Universal Robots PolyScope program: space invade.urp

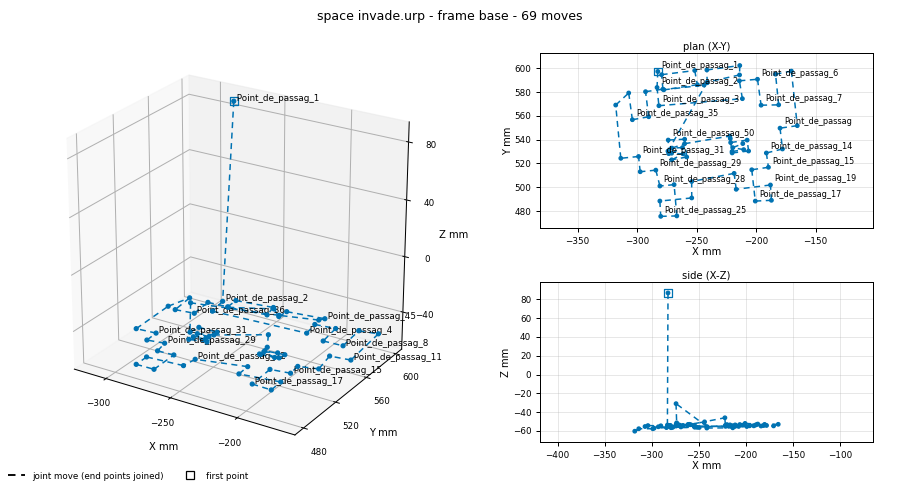
[picture p0: tool path of space invade.urp in frame base, 69 of 69 moves have a stored position in this frame; points joined in program order, loops and branches not executed]
ProgramRoot directory=/programs; kinematics=(a=[0, -0.425, -0.39225, 0, 0, 0], d=[0.08916, 0, 0, 0.10915, 0.09465, 0.0823], alpha=[1.5708, 0, 0, 1.5708, -1.5708, 0], deltaTheta=[0, 0, 0, 0, 0, 0], status=notInitialized); name=space invade; programVersion=(project__name=PolyScope, major__version=1, minor__version=6, svn__revision=9671, build__date=Dec 17 2012, 15:17:18); robotEnvironmentFileName=default
  MainProgram cartesianAcceleration=1.2; cartesianSpeed=0.25; jointAcceleration=1.3962634015954636; jointSpeed=1.0471975511965976; moveAsFastAsPossible=true; sharedProcessMoveBlendRadius=0.025; featureReference=(installationNameReference=Base); motionType=JOINT_SPACE
    Move cartesianAcceleration=1.2; cartesianSpeed=0.25; jointAcceleration=3.141592653589793; jointSpeed=3.2; moveAsFastAsPossible=true; sharedProcessMoveBlendRadius=0.025; featureReference=(installationNameReference=Base); motionType=JOINT_SPACE
      Waypoint blendRadius=0.05; cartesianAcceleration=1.2; cartesianSpeed=0.25; jointAcceleration=1.3962634015954636; jointSpeed=1.0471975511965976; nextMotionTime=2.0; stoppoint=true; useSharedBlendParameter=true; useSharedParameters=true; position=TCP in base x=-282.652 y=597.285 z=86.76 mm, rx=0.0179 ry=-1.8099 rz=-2.292 rad; joints [-73.183, -51.912, 94.402, -56.585, 97.955, 5.493] deg; positionType=FIXED_POSITION; waypointPoseInFeatureCoordinates=(pos=(x=-0.28265202221526026, y=0.5972847385628794, z=0.08675977077379672), rot=(x=0.017936265921650735, y=-1.8098588398059938, z=-2.292012778294841)); name=Point_de_passag_1
      Waypoint blendRadius=0.05; cartesianAcceleration=1.2; cartesianSpeed=0.25; jointAcceleration=1.3962634015954636; jointSpeed=1.0471975511965976; nextMotionTime=2.0; stoppoint=true; useSharedBlendParameter=true; useSharedParameters=true; position=TCP in base x=-283.288 y=583.825 z=-53.768 mm, rx=0.0625 ry=-2.0582 rz=-2.1165 rad; joints [-72.781, -39.176, 93.788, -56.699, 97.955, 5.493] deg; positionType=FIXED_POSITION; waypointPoseInFeatureCoordinates=(pos=(x=-0.2832877979734777, y=0.5838250260366411, z=-0.05376751381244214), rot=(x=0.062483678270235946, y=-2.0582415675415118, z=-2.1164651392423814)); name=Point_de_passag_2
      Waypoint blendRadius=0.05; cartesianAcceleration=1.2; cartesianSpeed=0.25; jointAcceleration=1.3962634015954636; jointSpeed=1.0471975511965976; nextMotionTime=2.0; stoppoint=true; useSharedBlendParameter=true; useSharedParameters=true; position=TCP in base x=-281.72 y=568.489 z=-54.598 mm, rx=0.0587 ry=-2.0396 rz=-2.1304 rad; joints [-72.458, -40.149, 96.768, -59.625, 98.3, 5.501] deg; positionType=FIXED_POSITION; waypointPoseInFeatureCoordinates=(pos=(x=-0.281720012954096, y=0.5684887438702723, z=-0.05459769912919604), rot=(x=0.058675556399115224, y=-2.0395702398943603, z=-2.13038736968013)); name=Point_de_passag_3
      Waypoint blendRadius=0.05; cartesianAcceleration=1.2; cartesianSpeed=0.25; jointAcceleration=1.3962634015954636; jointSpeed=1.0471975511965976; nextMotionTime=2.0; stoppoint=true; useSharedBlendParameter=true; useSharedParameters=true; position=TCP in base x=-211.543 y=574.409 z=-55.23 mm, rx=0.0579 ry=-2.0297 rz=-2.1391 rad; joints [-79.937, -41.862, 101.524, -63.144, 90.855, 5.884] deg; positionType=FIXED_POSITION; waypointPoseInFeatureCoordinates=(pos=(x=-0.21154341819000044, y=0.5744085042322971, z=-0.055229503778557475), rot=(x=0.057937704493810346, y=-2.0297402818102475, z=-2.1390769916078325)); name=Point_de_passag_4
      Waypoint blendRadius=0.05; cartesianAcceleration=1.2; cartesianSpeed=0.25; jointAcceleration=1.3962634015954636; jointSpeed=1.0471975511965976; nextMotionTime=2.0; stoppoint=true; useSharedBlendParameter=true; useSharedParameters=true; position=TCP in base x=-214.075 y=589.436 z=-55.719 mm, rx=0.0627 ry=-2.0275 rz=-2.1366 rad; joints [-79.992, -40.732, 98.758, -61.519, 90.535, 5.897] deg; positionType=FIXED_POSITION; waypointPoseInFeatureCoordinates=(pos=(x=-0.21407464423603903, y=0.5894359632457946, z=-0.05571947582978173), rot=(x=0.06269876874726125, y=-2.027465428705575, z=-2.136562643256111)); name=Point_de_passag_5
      Waypoint blendRadius=0.05; cartesianAcceleration=1.2; cartesianSpeed=0.25; jointAcceleration=1.3962634015954636; jointSpeed=1.0471975511965976; nextMotionTime=2.0; stoppoint=true; useSharedBlendParameter=true; useSharedParameters=true; position=TCP in base x=-198.843 y=590.725 z=-55.313 mm, rx=0.038 ry=-2.0446 rz=-2.1463 rad; joints [-81.41, -41.078, 99.401, -61.519, 90.535, 5.897] deg; positionType=FIXED_POSITION; waypointPoseInFeatureCoordinates=(pos=(x=-0.19884274831083149, y=0.5907248290980777, z=-0.05531313116339641), rot=(x=0.03796253245291551, y=-2.0446315901083487, z=-2.1462512241104803)); name=Point_de_passag_6
      Waypoint blendRadius=0.05; cartesianAcceleration=1.2; cartesianSpeed=0.25; jointAcceleration=1.3962634015954636; jointSpeed=1.0471975511965976; nextMotionTime=2.0; stoppoint=true; useSharedBlendParameter=true; useSharedParameters=true; position=TCP in base x=-195.825 y=568.935 z=-54.572 mm, rx=0.0394 ry=-2.0782 rz=-2.1171 rad; joints [-81.384, -42.82, 102.942, -61.605, 90.535, 5.897] deg; positionType=FIXED_POSITION; waypointPoseInFeatureCoordinates=(pos=(x=-0.19582460156289885, y=0.5689351016692715, z=-0.05457238838580761), rot=(x=0.03936187740158152, y=-2.0781510877701574, z=-2.117142621152102)); name=Point_de_passag_7
      Waypoint blendRadius=0.05; cartesianAcceleration=1.2; cartesianSpeed=0.25; jointAcceleration=1.3962634015954636; jointSpeed=1.0471975511965976; nextMotionTime=2.0; stoppoint=true; useSharedBlendParameter=true; useSharedParameters=true; position=TCP in base x=-181.043 y=569.228 z=-54.284 mm, rx=0.0462 ry=-2.0702 rz=-2.1187 rad; joints [-83.1, -43.176, 103.906, -62.493, 88.47, 5.923] deg; positionType=FIXED_POSITION; waypointPoseInFeatureCoordinates=(pos=(x=-0.1810427609560639, y=0.5692282541956158, z=-0.054283796649596934), rot=(x=0.04615435616599969, y=-2.0701592505685245, z=-2.118742154701426)); name=Point_de_passag_8
      Waypoint blendRadius=0.05; cartesianAcceleration=1.2; cartesianSpeed=0.25; jointAcceleration=1.3962634015954636; jointSpeed=1.0471975511965976; nextMotionTime=2.0; stoppoint=true; useSharedBlendParameter=true; useSharedParameters=true; position=TCP in base x=-183.68 y=594.979 z=-54.792 mm, rx=0.047 ry=-2.0708 rz=-2.1175 rad; joints [-83.158, -41.31, 99.23, -59.632, 88.371, 5.922] deg; positionType=FIXED_POSITION; waypointPoseInFeatureCoordinates=(pos=(x=-0.1836800661049113, y=0.594979301817125, z=-0.054791600611601515), rot=(x=0.04696593879286466, y=-2.070839020850319, z=-2.117502148687866)); name=Point_de_passag_9
      Waypoint blendRadius=0.05; cartesianAcceleration=1.2; cartesianSpeed=0.25; jointAcceleration=1.3962634015954636; jointSpeed=1.0471975511965976; nextMotionTime=2.0; stoppoint=true; useSharedBlendParameter=true; useSharedParameters=true; position=TCP in base x=-170.355 y=597.597 z=-54.676 mm, rx=0.0251 ry=-2.0908 rz=-2.1203 rad; joints [-84.434, -41.447, 99.329, -59.059, 88.304, 5.922] deg; positionType=FIXED_POSITION; waypointPoseInFeatureCoordinates=(pos=(x=-0.17035484047527763, y=0.597597198010664, z=-0.05467596987549106), rot=(x=0.025093825724090947, y=-2.0907687683588985, z=-2.120265521565159)); name=Point_de_passag_10
      Waypoint blendRadius=0.013000000000000001; cartesianAcceleration=1.2; cartesianSpeed=0.25; jointAcceleration=1.3962634015954636; jointSpeed=1.0471975511965976; nextMotionTime=2.0; useSharedParameters=true; position=TCP in base x=-165.398 y=551.726 z=-52.96 mm, rx=0.0232 ry=-2.1474 rz=-2.0682 rad; joints [-84.483, -45.032, 106.82, -60.011, 88.304, 5.922] deg; positionType=FIXED_POSITION; waypointPoseInFeatureCoordinates=(pos=(x=-0.16539794653699985, y=0.5517262593257032, z=-0.052959652162168705), rot=(x=0.023224151825996287, y=-2.1474477075993104, z=-2.0682381332856656)); name=Point_de_passag_11
      Waypoint blendRadius=0.05; cartesianAcceleration=1.2; cartesianSpeed=0.25; jointAcceleration=1.3962634015954636; jointSpeed=1.0471975511965976; nextMotionTime=2.0; stoppoint=true; useSharedBlendParameter=true; useSharedParameters=true; position=TCP in base x=-179.909 y=549.645 z=-53.069 mm, rx=0.0508 ry=-2.1312 rz=-2.0583 rad; joints [-83, -44.844, 106.464, -60.081, 88.303, 5.922] deg; positionType=FIXED_POSITION; waypointPoseInFeatureCoordinates=(pos=(x=-0.17990921422879388, y=0.5496453696656896, z=-0.05306886642297695), rot=(x=0.0507700070809368, y=-2.131176807810905, z=-2.058330386951994)); name=Point_de_passag
      Waypoint blendRadius=0.05; cartesianAcceleration=1.2; cartesianSpeed=0.25; jointAcceleration=1.3962634015954636; jointSpeed=1.0471975511965976; nextMotionTime=2.0; stoppoint=true; useSharedBlendParameter=true; useSharedParameters=true; position=TCP in base x=-177.842 y=532.133 z=-54.192 mm, rx=0.0511 ry=-2.0852 rz=-2.1006 rad; joints [-82.991, -45.659, 110.119, -65.332, 88.305, 5.922] deg; positionType=FIXED_POSITION; waypointPoseInFeatureCoordinates=(pos=(x=-0.1778422060960944, y=0.5321330621123782, z=-0.054192047949219516), rot=(x=0.051094345427341016, y=-2.085185673550667, z=-2.100645513934709)); name=Point_de_passag_13
      Waypoint blendRadius=0.05; cartesianAcceleration=1.2; cartesianSpeed=0.25; jointAcceleration=1.3962634015954636; jointSpeed=1.0471975511965976; nextMotionTime=2.0; stoppoint=true; useSharedBlendParameter=true; useSharedParameters=true; position=TCP in base x=-191.407 y=528.761 z=-54.614 mm, rx=0.077 ry=-2.0721 rz=-2.0875 rad; joints [-81.545, -45.517, 109.908, -65.34, 88.305, 5.922] deg; positionType=FIXED_POSITION; waypointPoseInFeatureCoordinates=(pos=(x=-0.19140661350513236, y=0.5287613442499617, z=-0.054613754535260246), rot=(x=0.076989872868353, y=-2.072075950982007, z=-2.0874887299160414)); name=Point_de_passag_14
      Waypoint blendRadius=0.05; cartesianAcceleration=1.2; cartesianSpeed=0.25; jointAcceleration=1.3962634015954636; jointSpeed=1.0471975511965976; nextMotionTime=2.0; stoppoint=true; useSharedBlendParameter=true; useSharedParameters=true; position=TCP in base x=-189.635 y=516.737 z=-53.772 mm, rx=0.0772 ry=-2.0943 rz=-2.0674 rad; joints [-81.544, -46.475, 111.695, -65.009, 88.305, 5.922] deg; positionType=FIXED_POSITION; waypointPoseInFeatureCoordinates=(pos=(x=-0.18963463358635635, y=0.516736619244103, z=-0.0537718213838417), rot=(x=0.07721179414043056, y=-2.0942602650848525, z=-2.0674493445746314)); name=Point_de_passag_15
      Waypoint blendRadius=0.05; cartesianAcceleration=1.2; cartesianSpeed=0.25; jointAcceleration=1.3962634015954636; jointSpeed=1.0471975511965976; nextMotionTime=2.0; stoppoint=true; useSharedBlendParameter=true; useSharedParameters=true; position=TCP in base x=-203.672 y=514.674 z=-53.972 mm, rx=0.1039 ry=-2.0705 rz=-2.0627 rad; joints [-80.04, -46.204, 111.312, -65.495, 88.305, 5.922] deg; positionType=FIXED_POSITION; waypointPoseInFeatureCoordinates=(pos=(x=-0.20367177630866146, y=0.5146735620035543, z=-0.05397197974529697), rot=(x=0.1038793388777256, y=-2.0705290115638433, z=-2.062731628632467)); name=Point_de_passag_16
      Waypoint blendRadius=0.05; cartesianAcceleration=1.2; cartesianSpeed=0.25; jointAcceleration=1.3962634015954636; jointSpeed=1.0471975511965976; nextMotionTime=2.0; stoppoint=true; useSharedBlendParameter=true; useSharedParameters=true; position=TCP in base x=-200.707 y=488.328 z=-52.009 mm, rx=0.1082 ry=-2.1145 rz=-2.0196 rad; joints [-79.858, -48.24, 115.109, -64.859, 88.305, 5.922] deg; positionType=FIXED_POSITION; waypointPoseInFeatureCoordinates=(pos=(x=-0.20070659319109455, y=0.48832793802061364, z=-0.05200930305093718), rot=(x=0.1081532575906928, y=-2.114489458793282, z=-2.0196190971781767)); name=Point_de_passag_17
      Waypoint blendRadius=0.05; cartesianAcceleration=1.2; cartesianSpeed=0.25; jointAcceleration=1.3962634015954636; jointSpeed=1.0471975511965976; nextMotionTime=2.0; stoppoint=true; useSharedBlendParameter=true; useSharedParameters=true; position=TCP in base x=-187.143 y=488.994 z=-52.712 mm, rx=0.0809 ry=-2.1346 rz=-2.0269 rad; joints [-81.363, -48.441, 115.733, -64.867, 88.305, 5.922] deg; positionType=FIXED_POSITION; waypointPoseInFeatureCoordinates=(pos=(x=-0.1871430029431406, y=0.48899418849543297, z=-0.05271155794650809), rot=(x=0.08088198197152559, y=-2.1346176021906746, z=-2.026919975113168)); name=Point_de_passag_18
      Waypoint blendRadius=0.05; cartesianAcceleration=1.2; cartesianSpeed=0.25; jointAcceleration=1.3962634015954636; jointSpeed=1.0471975511965976; nextMotionTime=2.0; stoppoint=true; useSharedBlendParameter=true; useSharedParameters=true; position=TCP in base x=-187.962 y=501.873 z=-52.995 mm, rx=0.0784 ry=-2.114 rz=-2.0483 rad; joints [-81.486, -47.562, 113.928, -65.089, 88.305, 5.922] deg; positionType=FIXED_POSITION; waypointPoseInFeatureCoordinates=(pos=(x=-0.1879615483845748, y=0.5018733241174247, z=-0.05299473152099478), rot=(x=0.07843748330968311, y=-2.114018702598733, z=-2.0482981478056983)); name=Point_de_passag_19
      Waypoint blendRadius=0.05; cartesianAcceleration=1.2; cartesianSpeed=0.25; jointAcceleration=1.3962634015954636; jointSpeed=1.0471975511965976; nextMotionTime=2.0; stoppoint=true; useSharedBlendParameter=true; useSharedParameters=true; position=TCP in base x=-216.735 y=498.237 z=-53.591 mm, rx=0.134 ry=-2.0632 rz=-2.0396 rad; joints [-78.342, -46.912, 112.982, -66.105, 88.306, 5.922] deg; positionType=FIXED_POSITION; waypointPoseInFeatureCoordinates=(pos=(x=-0.21673546092603405, y=0.4982370374973547, z=-0.05359079206576065), rot=(x=0.1339840578207861, y=-2.063161429904662, z=-2.039595644626832)); name=Point_de_passag_20
      Waypoint blendRadius=0.05; cartesianAcceleration=1.2; cartesianSpeed=0.25; jointAcceleration=1.3962634015954636; jointSpeed=1.0471975511965976; nextMotionTime=2.0; stoppoint=true; useSharedBlendParameter=true; useSharedParameters=true; position=TCP in base x=-218.491 y=511.628 z=-54.705 mm, rx=0.1314 ry=-2.0424 rz=-2.0596 rad; joints [-78.446, -45.862, 111.005, -66.308, 88.305, 5.922] deg; positionType=FIXED_POSITION; waypointPoseInFeatureCoordinates=(pos=(x=-0.21849083751855686, y=0.5116284107631719, z=-0.05470477091723423), rot=(x=0.13139877328918678, y=-2.0424162115946194, z=-2.05961440507516)); name=Point_de_passag_21
      Waypoint blendRadius=0.05; cartesianAcceleration=1.2; cartesianSpeed=0.25; jointAcceleration=1.3962634015954636; jointSpeed=1.0471975511965976; nextMotionTime=2.0; stoppoint=true; useSharedBlendParameter=true; useSharedParameters=true; position=TCP in base x=-254.179 y=504.815 z=-56.099 mm, rx=0.1932 ry=-1.9671 rz=-2.0561 rad; joints [-74.661, -44.909, 109.98, -68.477, 88.302, 5.922] deg; positionType=FIXED_POSITION; waypointPoseInFeatureCoordinates=(pos=(x=-0.25417942033963226, y=0.5048153116990209, z=-0.056099214267682045), rot=(x=0.19321471885735442, y=-1.9671482174053354, z=-2.056099784005873)); name=Point_de_passag_22
      Waypoint blendRadius=0.05; cartesianAcceleration=1.2; cartesianSpeed=0.25; jointAcceleration=1.3962634015954636; jointSpeed=1.0471975511965976; nextMotionTime=2.0; stoppoint=true; useSharedBlendParameter=true; useSharedParameters=true; position=TCP in base x=-254.115 y=490.968 z=-54.665 mm, rx=0.2009 ry=-1.9836 rz=-2.0358 rad; joints [-74.28, -45.959, 111.906, -68.331, 88.302, 5.922] deg; positionType=FIXED_POSITION; waypointPoseInFeatureCoordinates=(pos=(x=-0.25411498173780606, y=0.49096791980041576, z=-0.05466495035963062), rot=(x=0.2009396797645236, y=-1.9836045819608157, z=-2.0357660094942114)); name=Point_de_passag_23
      Waypoint blendRadius=0.05; cartesianAcceleration=1.2; cartesianSpeed=0.25; jointAcceleration=1.3962634015954636; jointSpeed=1.0471975511965976; nextMotionTime=2.0; stoppoint=true; useSharedBlendParameter=true; useSharedParameters=true; position=TCP in base x=-280.907 y=488.374 z=-54.511 mm, rx=0.2462 ry=-1.9581 rz=-2.0072 rad; joints [-71.517, -45.323, 110.098, -67.236, 88.302, 5.922] deg; positionType=FIXED_POSITION; waypointPoseInFeatureCoordinates=(pos=(x=-0.28090733276783925, y=0.48837398030980983, z=-0.05451080053554329), rot=(x=0.24622420703531242, y=-1.958097985487623, z=-2.007158780897492)); name=Point_de_passag_24
      Waypoint blendRadius=0.05; cartesianAcceleration=1.2; cartesianSpeed=0.25; jointAcceleration=1.3962634015954636; jointSpeed=1.0471975511965976; nextMotionTime=2.0; stoppoint=true; useSharedBlendParameter=true; useSharedParameters=true; position=TCP in base x=-280.183 y=475.501 z=-54.091 mm, rx=0.2537 ry=-1.9716 rz=-1.9896 rad; joints [-71.157, -46.173, 111.884, -67.298, 88.302, 5.922] deg; positionType=FIXED_POSITION; waypointPoseInFeatureCoordinates=(pos=(x=-0.2801828103663585, y=0.4755011085108045, z=-0.05409137347930281), rot=(x=0.25374819947138966, y=-1.971603919125501, z=-1.9896410426914868)); name=Point_de_passag_25
      Waypoint blendRadius=0.05; cartesianAcceleration=1.2; cartesianSpeed=0.25; jointAcceleration=1.3962634015954636; jointSpeed=1.0471975511965976; nextMotionTime=2.0; stoppoint=true; useSharedBlendParameter=true; useSharedParameters=true; position=TCP in base x=-266.657 y=475.862 z=-54.138 mm, rx=0.2303 ry=-1.9759 rz=-2.011 rad; joints [-72.54, -46.512, 113.086, -68.572, 88.302, 5.922] deg; positionType=FIXED_POSITION; waypointPoseInFeatureCoordinates=(pos=(x=-0.26665659194596086, y=0.4758620876423463, z=-0.05413763323845962), rot=(x=0.2303206574748975, y=-1.9759213595413552, z=-2.0109717755054826)); name=Point_de_passag_26
      Waypoint blendRadius=0.05; cartesianAcceleration=1.2; cartesianSpeed=0.25; jointAcceleration=1.3962634015954636; jointSpeed=1.0471975511965976; nextMotionTime=2.0; stoppoint=true; useSharedBlendParameter=true; useSharedParameters=true; position=TCP in base x=-268.941 y=502.155 z=-55.766 mm, rx=0.2178 ry=-1.9463 rz=-2.0455 rad; joints [-73.125, -44.635, 109.305, -68.468, 88.301, 5.922] deg; positionType=FIXED_POSITION; waypointPoseInFeatureCoordinates=(pos=(x=-0.2689413685160755, y=0.5021549803735984, z=-0.055766494413654645), rot=(x=0.21778406161377237, y=-1.9463059097964963, z=-2.045536292220743)); name=Point_de_passag_27
      Waypoint blendRadius=0.05; cartesianAcceleration=1.2; cartesianSpeed=0.25; jointAcceleration=1.3962634015954636; jointSpeed=1.0471975511965976; nextMotionTime=2.0; stoppoint=true; useSharedBlendParameter=true; useSharedParameters=true; position=TCP in base x=-280.879 y=500.999 z=-55.493 mm, rx=0.2363 ry=-1.9272 rz=-2.0393 rad; joints [-71.926, -44.328, 108.589, -68.509, 88.301, 5.922] deg; positionType=FIXED_POSITION; waypointPoseInFeatureCoordinates=(pos=(x=-0.28087883185661877, y=0.5009989517749368, z=-0.05549299786774024), rot=(x=0.2363220852941244, y=-1.9272014382031044, z=-2.03927583997445)); name=Point_de_passag_28
      Waypoint blendRadius=0.05; cartesianAcceleration=1.2; cartesianSpeed=0.25; jointAcceleration=1.3962634015954636; jointSpeed=1.0471975511965976; nextMotionTime=2.0; stoppoint=true; useSharedBlendParameter=true; useSharedParameters=true; position=TCP in base x=-284.3 y=514.345 z=-56.483 mm, rx=0.233 ry=-1.9076 rz=-2.0562 rad; joints [-72.015, -43.245, 106.46, -68.509, 88.301, 5.922] deg; positionType=FIXED_POSITION; waypointPoseInFeatureCoordinates=(pos=(x=-0.2842996140558753, y=0.5143447912365959, z=-0.0564829134063703), rot=(x=0.23300302579211407, y=-1.9076264084877625, z=-2.056223159122742)); name=Point_de_passag_29
      Waypoint blendRadius=0.05; cartesianAcceleration=1.2; cartesianSpeed=0.25; jointAcceleration=1.3962634015954636; jointSpeed=1.0471975511965976; nextMotionTime=2.0; stoppoint=true; useSharedBlendParameter=true; useSharedParameters=true; position=TCP in base x=-297.442 y=512.995 z=-57.051 mm, rx=0.252 ry=-1.8866 rz=-2.0495 rad; joints [-70.741, -42.778, 105.621, -68.645, 88.301, 5.922] deg; positionType=FIXED_POSITION; waypointPoseInFeatureCoordinates=(pos=(x=-0.2974424195632888, y=0.5129950839083096, z=-0.057050738658507585), rot=(x=0.2520285596450359, y=-1.8866198016302187, z=-2.049532572559801)); name=Point_de_passag_30
      Waypoint blendRadius=0.05; cartesianAcceleration=1.2; cartesianSpeed=0.25; jointAcceleration=1.3962634015954636; jointSpeed=1.0471975511965976; nextMotionTime=2.0; stoppoint=true; useSharedBlendParameter=true; useSharedParameters=true; position=TCP in base x=-298.817 y=525.813 z=-57.672 mm, rx=0.2461 ry=-1.8738 rz=-2.0644 rad; joints [-71.023, -41.845, 103.666, -68.404, 88.301, 5.922] deg; positionType=FIXED_POSITION; waypointPoseInFeatureCoordinates=(pos=(x=-0.2988172166861918, y=0.5258127782720562, z=-0.05767229073573248), rot=(x=0.2460544276065498, y=-1.873832889851444, z=-2.0643544978907182)); name=Point_de_passag_31
      Waypoint blendRadius=0.05; cartesianAcceleration=1.2; cartesianSpeed=0.25; jointAcceleration=1.3962634015954636; jointSpeed=1.0471975511965976; nextMotionTime=2.0; stoppoint=true; useSharedBlendParameter=true; useSharedParameters=true; position=TCP in base x=-313.744 y=524.322 z=-57.659 mm, rx=0.2662 ry=-1.8502 rz=-2.057 rad; joints [-69.627, -41.369, 102.67, -68.471, 88.301, 5.922] deg; positionType=FIXED_POSITION; waypointPoseInFeatureCoordinates=(pos=(x=-0.31374382039765136, y=0.5243217642102161, z=-0.05765907958066508), rot=(x=0.26623481915853003, y=-1.8501630766307802, z=-2.0569536481156736)); name=Point_de_passag_32
      Waypoint blendRadius=0.05; cartesianAcceleration=1.2; cartesianSpeed=0.25; jointAcceleration=1.3962634015954636; jointSpeed=1.0471975511965976; nextMotionTime=2.0; stoppoint=true; useSharedBlendParameter=true; useSharedParameters=true; position=TCP in base x=-318.02 y=569.053 z=-60.302 mm, rx=0.2432 ry=-1.7914 rz=-2.1182 rad; joints [-70.657, -37.847, 95.752, -68.493, 88.303, 5.922] deg; positionType=FIXED_POSITION; waypointPoseInFeatureCoordinates=(pos=(x=-0.3180203016728063, y=0.5690529321818526, z=-0.06030228769300152), rot=(x=0.24322621053901108, y=-1.7914029699628753, z=-2.118190938669368)); name=Point_de_passag_33
      Waypoint blendRadius=0.05; cartesianAcceleration=1.2; cartesianSpeed=0.25; jointAcceleration=1.3962634015954636; jointSpeed=1.0471975511965976; nextMotionTime=2.0; stoppoint=true; useSharedBlendParameter=true; useSharedParameters=true; position=TCP in base x=-307.099 y=579.197 z=-55.323 mm, rx=0.2377 ry=-1.9321 rz=-2.0344 rad; joints [-71.867, -38.625, 93.559, -58.906, 88.304, 5.922] deg; positionType=FIXED_POSITION; waypointPoseInFeatureCoordinates=(pos=(x=-0.30709884957894884, y=0.5791966633506883, z=-0.05532276369273085), rot=(x=0.23771813579159426, y=-1.9320563641421478, z=-2.034419190129147)); name=Point_de_passag_34
      Waypoint blendRadius=0.05; cartesianAcceleration=1.2; cartesianSpeed=0.25; jointAcceleration=1.3962634015954636; jointSpeed=1.0471975511965976; nextMotionTime=2.0; stoppoint=true; useSharedBlendParameter=true; useSharedParameters=true; position=TCP in base x=-304.023 y=556.724 z=-54.333 mm, rx=0.247 ry=-1.962 rz=-2.0036 rad; joints [-71.493, -40.465, 97.195, -58.975, 88.303, 5.922] deg; positionType=FIXED_POSITION; waypointPoseInFeatureCoordinates=(pos=(x=-0.30402280640175033, y=0.5567238167970993, z=-0.05433296925638692), rot=(x=0.24699226951245087, y=-1.9620119020797953, z=-2.0035693049412804)); name=Point_de_passag_35
      Waypoint blendRadius=0.05; cartesianAcceleration=1.2; cartesianSpeed=0.25; jointAcceleration=1.3962634015954636; jointSpeed=1.0471975511965976; nextMotionTime=2.0; stoppoint=true; useSharedBlendParameter=true; useSharedParameters=true; position=TCP in base x=-290.285 y=559.229 z=-54.533 mm, rx=0.2268 ry=-1.9808 rz=-2.0111 rad; joints [-72.768, -40.783, 97.886, -58.951, 88.303, 5.922] deg; positionType=FIXED_POSITION; waypointPoseInFeatureCoordinates=(pos=(x=-0.2902847442816515, y=0.5592288861188497, z=-0.05453277295753601), rot=(x=0.22679121942018315, y=-1.9808056849918738, z=-2.011055406226187)); name=Point_de_passag_36
      Waypoint blendRadius=0.05; cartesianAcceleration=1.2; cartesianSpeed=0.25; jointAcceleration=1.3962634015954636; jointSpeed=1.0471975511965976; nextMotionTime=2.0; stoppoint=true; useSharedBlendParameter=true; useSharedParameters=true; position=TCP in base x=-292.95 y=580.3 z=-55.604 mm, rx=0.2172 ry=-1.935 rz=-2.0542 rad; joints [-73.098, -39.003, 94.73, -60.1, 88.304, 5.922] deg; positionType=FIXED_POSITION; waypointPoseInFeatureCoordinates=(pos=(x=-0.2929495974619331, y=0.5803004815752308, z=-0.05560445383124647), rot=(x=0.21721197861069477, y=-1.9349740722438789, z=-2.0541876118542177)); name=Point_de_passag_37
      Waypoint blendRadius=0.05; cartesianAcceleration=1.2; cartesianSpeed=0.25; jointAcceleration=1.3962634015954636; jointSpeed=1.0471975511965976; nextMotionTime=2.0; stoppoint=true; useSharedBlendParameter=true; useSharedParameters=true; position=TCP in base x=-278.357 y=582.397 z=-56.119 mm, rx=0.1966 ry=-1.9548 rz=-2.0617 rad; joints [-74.409, -39.321, 95.48, -60.09, 88.303, 5.922] deg; positionType=FIXED_POSITION; waypointPoseInFeatureCoordinates=(pos=(x=-0.27835666891726796, y=0.5823967370196382, z=-0.05611873503618645), rot=(x=0.1965997085054426, y=-1.9548269218518175, z=-2.061655407008621)); name=Point_de_passag_38
      Waypoint blendRadius=0.05; cartesianAcceleration=1.2; cartesianSpeed=0.25; jointAcceleration=1.3962634015954636; jointSpeed=1.0471975511965976; nextMotionTime=2.0; stoppoint=true; useSharedBlendParameter=true; useSharedParameters=true; position=TCP in base x=-279.428 y=594.592 z=-56.586 mm, rx=0.1919 ry=-1.9364 rz=-2.08 rad; joints [-74.608, -38.322, 93.522, -60.161, 88.303, 5.922] deg; positionType=FIXED_POSITION; waypointPoseInFeatureCoordinates=(pos=(x=-0.27942759926614935, y=0.5945918660928576, z=-0.05658591167334987), rot=(x=0.19192313364052163, y=-1.9364372193914225, z=-2.0799532137280012)); name=Point_de_passag_39
      Waypoint blendRadius=0.05; cartesianAcceleration=1.2; cartesianSpeed=0.25; jointAcceleration=1.3962634015954636; jointSpeed=1.0471975511965976; nextMotionTime=2.0; stoppoint=true; useSharedBlendParameter=true; useSharedParameters=true; position=TCP in base x=-251.594 y=598.088 z=-56.2 mm, rx=0.1518 ry=-1.9684 rz=-2.0981 rad; joints [-77.088, -39.028, 94.956, -60.326, 88.303, 5.922] deg; positionType=FIXED_POSITION; waypointPoseInFeatureCoordinates=(pos=(x=-0.2515935489777176, y=0.5980877570075677, z=-0.05620023801837448), rot=(x=0.15184243528629326, y=-1.9684070112876602, z=-2.0981215006048926)); name=Point_de_passag_40
      Waypoint blendRadius=0.05; cartesianAcceleration=1.2; cartesianSpeed=0.25; jointAcceleration=1.3962634015954636; jointSpeed=1.0471975511965976; nextMotionTime=2.0; stoppoint=true; useSharedBlendParameter=true; useSharedParameters=true; position=TCP in base x=-249.398 y=586.161 z=-56.31 mm, rx=0.1533 ry=-1.9809 rz=-2.087 rad; joints [-77.04, -39.954, 97.045, -60.829, 88.303, 5.922] deg; positionType=FIXED_POSITION; waypointPoseInFeatureCoordinates=(pos=(x=-0.24939827566667166, y=0.5861607728670549, z=-0.05631023731002235), rot=(x=0.15327321649812645, y=-1.9808671189960518, z=-2.0870336376894985)); name=Point_de_passag_41
      Waypoint blendRadius=0.05; cartesianAcceleration=1.2; cartesianSpeed=0.25; jointAcceleration=1.3962634015954636; jointSpeed=1.0471975511965976; nextMotionTime=2.0; stoppoint=true; useSharedBlendParameter=true; useSharedParameters=true; position=TCP in base x=-277.574 y=581.867 z=-56.086 mm, rx=0.1946 ry=-1.9392 rz=-2.0754 rad; joints [-74.464, -39.337, 95.853, -61.278, 88.309, 5.914] deg; positionType=FIXED_POSITION; waypointPoseInFeatureCoordinates=(pos=(x=-0.27757359218810485, y=0.5818667372671205, z=-0.05608584955968336), rot=(x=0.1945895499015074, y=-1.9391807919038222, z=-2.075415897091717)); name=Point_de_passag_60
      Waypoint blendRadius=0.05; cartesianAcceleration=1.2; cartesianSpeed=0.25; jointAcceleration=1.3962634015954636; jointSpeed=1.0471975511965976; nextMotionTime=2.0; stoppoint=true; useSharedBlendParameter=true; useSharedParameters=true; position=TCP in base x=-243.779 y=585.859 z=-50.341 mm, rx=0.1452 ry=-1.9912 rz=-2.0872 rad; joints [-77.536, -40.838, 97.537, -60.12, 88.303, 5.922] deg; positionType=FIXED_POSITION; waypointPoseInFeatureCoordinates=(pos=(x=-0.24377938935960666, y=0.5858590392549986, z=-0.05034104395441085), rot=(x=0.14523607646899533, y=-1.9912020479433818, z=-2.087198891102561)); name=Point_de_passag_42
      Waypoint blendRadius=0.05; cartesianAcceleration=1.2; cartesianSpeed=0.25; jointAcceleration=1.3962634015954636; jointSpeed=1.0471975511965976; nextMotionTime=2.0; stoppoint=true; useSharedBlendParameter=true; useSharedParameters=true; position=TCP in base x=-241.133 y=587.802 z=-56.085 mm, rx=0.1408 ry=-1.9991 rz=-2.0854 rad; joints [-77.811, -40.141, 97.207, -60.198, 88.303, 5.922] deg; positionType=FIXED_POSITION; waypointPoseInFeatureCoordinates=(pos=(x=-0.24113262365099739, y=0.5878017256628483, z=-0.056084920870279456), rot=(x=0.14083167022710746, y=-1.9991211656115546, z=-2.0854201544661213)); name=Point_de_passag_43
      Waypoint blendRadius=0.05; cartesianAcceleration=1.2; cartesianSpeed=0.25; jointAcceleration=1.3962634015954636; jointSpeed=1.0471975511965976; nextMotionTime=2.0; stoppoint=true; useSharedBlendParameter=true; useSharedParameters=true; position=TCP in base x=-241.389 y=598.571 z=-56.938 mm, rx=0.1355 ry=-1.9464 rz=-2.1319 rad; joints [-77.993, -39.11, 95.983, -62.774, 88.303, 5.922] deg; positionType=FIXED_POSITION; waypointPoseInFeatureCoordinates=(pos=(x=-0.2413893701404747, y=0.5985710803716395, z=-0.056938060225692845), rot=(x=0.1355239293187668, y=-1.9463810334033986, z=-2.131911015250782)); name=Point_de_passag_44
      Waypoint blendRadius=0.05; cartesianAcceleration=1.2; cartesianSpeed=0.25; jointAcceleration=1.3962634015954636; jointSpeed=1.0471975511965976; nextMotionTime=2.0; stoppoint=true; useSharedBlendParameter=true; useSharedParameters=true; position=TCP in base x=-213.756 y=602.278 z=-56.686 mm, rx=0.0941 ry=-1.9984 rz=-2.1333 rad; joints [-80.515, -39.72, 96.791, -61.379, 88.303, 5.922] deg; positionType=FIXED_POSITION; waypointPoseInFeatureCoordinates=(pos=(x=-0.21375646991851008, y=0.6022783347738264, z=-0.05668610917157056), rot=(x=0.09410599137776675, y=-1.9984416074849614, z=-2.13333212074026)); name=Point_de_passag_45
      Waypoint blendRadius=0.05; cartesianAcceleration=1.2; cartesianSpeed=0.25; jointAcceleration=1.3962634015954636; jointSpeed=1.0471975511965976; nextMotionTime=2.0; stoppoint=true; useSharedBlendParameter=true; useSharedParameters=true; position=TCP in base x=-213.921 y=594.364 z=-54.462 mm, rx=0.0979 ry=-2.0752 rz=-2.0644 rad; joints [-80.38, -40.74, 97.151, -56.699, 88.303, 5.922] deg; positionType=FIXED_POSITION; waypointPoseInFeatureCoordinates=(pos=(x=-0.21392060063374338, y=0.5943643098109264, z=-0.054462330208542846), rot=(x=0.09792232311371865, y=-2.075214898947158, z=-2.064431460289385)); name=Point_de_passag_46
      Waypoint blendRadius=0.05; cartesianAcceleration=1.2; cartesianSpeed=0.25; jointAcceleration=1.3962634015954636; jointSpeed=1.0471975511965976; nextMotionTime=2.0; stoppoint=true; useSharedBlendParameter=true; useSharedParameters=true; position=TCP in base x=-241.144 y=588.34 z=-55.468 mm, rx=0.141 ry=-2.0062 rz=-2.0796 rad; joints [-77.82, -40.194, 97.028, -59.604, 88.303, 5.922] deg; positionType=FIXED_POSITION; waypointPoseInFeatureCoordinates=(pos=(x=-0.24114357466003372, y=0.5883396110274949, z=-0.05546753961388532), rot=(x=0.14096730037012506, y=-2.006216665072978, z=-2.079615420375156)); name=Point_de_passag_47
      Waypoint blendRadius=0.05; cartesianAcceleration=1.2; cartesianSpeed=0.25; jointAcceleration=1.3962634015954636; jointSpeed=1.0471975511965976; nextMotionTime=2.0; stoppoint=true; useSharedBlendParameter=true; useSharedParameters=true; position=TCP in base x=-274.108 y=530.294 z=-31.01 mm, rx=0.221 ry=-2.0526 rz=-1.9618 rad; joints [-73.44, -46.153, 103.354, -55.57, 88.3, 5.922] deg; positionType=FIXED_POSITION; waypointPoseInFeatureCoordinates=(pos=(x=-0.2741078900677437, y=0.5302942442847837, z=-0.031009507499449487), rot=(x=0.22100803224921625, y=-2.052621942977806, z=-1.9618407208571134)); name=Point_de_passag_48
      Waypoint blendRadius=0.05; cartesianAcceleration=1.2; cartesianSpeed=0.25; jointAcceleration=1.3962634015954636; jointSpeed=1.0471975511965976; nextMotionTime=2.0; stoppoint=true; useSharedBlendParameter=true; useSharedParameters=true; position=TCP in base x=-273.441 y=528.214 z=-51.379 mm, rx=0.2236 ry=-2.0863 rz=-1.9319 rad; joints [-73.444, -43.981, 102.989, -55.571, 88.3, 5.922] deg; positionType=FIXED_POSITION; waypointPoseInFeatureCoordinates=(pos=(x=-0.27344084871747437, y=0.5282139416916622, z=-0.051378738040547364), rot=(x=0.22360964219232346, y=-2.0863408661862177, z=-1.9318784697090337)); name=Point_de_passag_49
      Waypoint blendRadius=0.05; cartesianAcceleration=1.2; cartesianSpeed=0.25; jointAcceleration=1.3962634015954636; jointSpeed=1.0471975511965976; nextMotionTime=2.0; stoppoint=true; useSharedBlendParameter=true; useSharedParameters=true; position=TCP in base x=-273.883 y=539.651 z=-52.715 mm, rx=0.2152 ry=-2.0424 rz=-1.9757 rad; joints [-73.717, -42.97, 101.778, -57.848, 88.301, 5.922] deg; positionType=FIXED_POSITION; waypointPoseInFeatureCoordinates=(pos=(x=-0.27388273515686756, y=0.5396508503812484, z=-0.05271466776412062), rot=(x=0.21524376014662439, y=-2.04241925853219, z=-1.9757460249285042)); name=Point_de_passag_50
      Waypoint blendRadius=0.05; cartesianAcceleration=1.2; cartesianSpeed=0.25; jointAcceleration=1.3962634015954636; jointSpeed=1.0471975511965976; nextMotionTime=2.0; stoppoint=true; useSharedBlendParameter=true; useSharedParameters=true; position=TCP in base x=-260.069 y=540.339 z=-52.981 mm, rx=0.1926 ry=-2.0477 rz=-1.9943 rad; joints [-75.024, -43.319, 102.869, -58.911, 88.291, 5.922] deg; positionType=FIXED_POSITION; waypointPoseInFeatureCoordinates=(pos=(x=-0.2600694702676959, y=0.5403391968339236, z=-0.052980628015052066), rot=(x=0.19255344037769048, y=-2.0476516084548306, z=-1.9943262347789312)); name=Point_de_passag_51
      Waypoint blendRadius=0.05; cartesianAcceleration=1.2; cartesianSpeed=0.25; jointAcceleration=1.3962634015954636; jointSpeed=1.0471975511965976; nextMotionTime=2.0; stoppoint=true; useSharedBlendParameter=true; useSharedParameters=true; position=TCP in base x=-258.347 y=525.385 z=-53.434 mm, rx=0.1966 ry=-2.0497 rz=-1.9887 rad; joints [-74.805, -44.271, 105.373, -60.255, 88.291, 5.922] deg; positionType=FIXED_POSITION; waypointPoseInFeatureCoordinates=(pos=(x=-0.25834723893751077, y=0.5253847483282241, z=-0.05343432663687591), rot=(x=0.1965938421441596, y=-2.049664497835512, z=-1.9886565144535326)); name=Point_de_passag_52
      Waypoint blendRadius=0.05; cartesianAcceleration=1.2; cartesianSpeed=0.25; jointAcceleration=1.3962634015954636; jointSpeed=1.0471975511965976; nextMotionTime=2.0; stoppoint=true; useSharedBlendParameter=true; useSharedParameters=true; position=TCP in base x=-270.942 y=523.013 z=-53.785 mm, rx=0.2166 ry=-2.0169 rz=-1.9943 rad; joints [-73.536, -43.911, 105.036, -61.425, 88.291, 5.922] deg; positionType=FIXED_POSITION; waypointPoseInFeatureCoordinates=(pos=(x=-0.270942258439706, y=0.5230127472168813, z=-0.053784779111683584), rot=(x=0.21661661673267862, y=-2.0169147781772665, z=-1.9942978127943105)); name=Point_de_passag_53
      Waypoint blendRadius=0.05; cartesianAcceleration=1.2; cartesianSpeed=0.25; jointAcceleration=1.3962634015954636; jointSpeed=1.0471975511965976; nextMotionTime=2.0; stoppoint=true; useSharedBlendParameter=true; useSharedParameters=true; position=TCP in base x=-261.275 y=528.016 z=-53.142 mm, rx=0.1984 ry=-2.0246 rz=-2.0071 rad; joints [-74.589, -43.977, 105.053, -61.469, 88.316, 5.914] deg; positionType=FIXED_POSITION; waypointPoseInFeatureCoordinates=(pos=(x=-0.26127468790307845, y=0.5280155272441636, z=-0.05314182227724498), rot=(x=0.19837290862743964, y=-2.024567289756419, z=-2.0071464871603557)); name=Point_de_passag_66
      Waypoint blendRadius=0.05; cartesianAcceleration=1.2; cartesianSpeed=0.25; jointAcceleration=1.3962634015954636; jointSpeed=1.0471975511965976; nextMotionTime=2.0; stoppoint=true; useSharedBlendParameter=true; useSharedParameters=true; position=TCP in base x=-271.039 y=528.559 z=-54.292 mm, rx=0.2135 ry=-2.0125 rz=-2.0012 rad; joints [-73.678, -43.486, 104.212, -61.339, 88.316, 5.914] deg; positionType=FIXED_POSITION; waypointPoseInFeatureCoordinates=(pos=(x=-0.2710392223663191, y=0.5285590376057627, z=-0.05429231420522969), rot=(x=0.21348299907923818, y=-2.0124902277950065, z=-2.0011703545267294)); name=Point_de_passag_67
      Waypoint blendRadius=0.05; cartesianAcceleration=1.2; cartesianSpeed=0.25; jointAcceleration=1.3962634015954636; jointSpeed=1.0471975511965976; nextMotionTime=2.0; stoppoint=true; useSharedBlendParameter=true; useSharedParameters=true; position=TCP in base x=-261.877 y=533.291 z=-53.779 mm, rx=0.1966 ry=-2.0202 rz=-2.0123 rad; joints [-74.67, -43.537, 104.212, -61.335, 88.316, 5.914] deg; positionType=FIXED_POSITION; waypointPoseInFeatureCoordinates=(pos=(x=-0.2618766895856911, y=0.5332907055387588, z=-0.0537790138928185), rot=(x=0.19664944376242535, y=-2.020191213780406, z=-2.0123274984489683)); name=Point_de_passag_68
      Waypoint blendRadius=0.05; cartesianAcceleration=1.2; cartesianSpeed=0.25; jointAcceleration=1.3962634015954636; jointSpeed=1.0471975511965976; nextMotionTime=2.0; stoppoint=true; useSharedBlendParameter=true; useSharedParameters=true; position=TCP in base x=-270.751 y=532.861 z=-53.724 mm, rx=0.2105 ry=-2.0071 rz=-2.0084 rad; joints [-73.822, -43.274, 103.646, -61.335, 88.317, 5.914] deg; positionType=FIXED_POSITION; waypointPoseInFeatureCoordinates=(pos=(x=-0.2707513479987141, y=0.5328613225686027, z=-0.05372435777231338), rot=(x=0.21051183542041538, y=-2.0070608181730125, z=-2.0083723043569637)); name=Point_de_passag_69
      Waypoint blendRadius=0.05; cartesianAcceleration=1.2; cartesianSpeed=0.25; jointAcceleration=1.3962634015954636; jointSpeed=1.0471975511965976; nextMotionTime=2.0; stoppoint=true; useSharedBlendParameter=true; useSharedParameters=true; position=TCP in base x=-260.137 y=536.557 z=-53.439 mm, rx=0.192 ry=-2.0173 rz=-2.0193 rad; joints [-74.918, -43.409, 103.896, -61.412, 88.319, 5.914] deg; positionType=FIXED_POSITION; waypointPoseInFeatureCoordinates=(pos=(x=-0.26013669014201773, y=0.5365565428164334, z=-0.0534394755675335), rot=(x=0.19203063200739287, y=-2.017262736006623, z=-2.019278237405916)); name=Point_de_passag_70
      Waypoint blendRadius=0.05; cartesianAcceleration=1.2; cartesianSpeed=0.25; jointAcceleration=1.3962634015954636; jointSpeed=1.0471975511965976; nextMotionTime=2.0; stoppoint=true; useSharedBlendParameter=true; useSharedParameters=true; position=TCP in base x=-222.133 y=542.993 z=-46.02 mm, rx=0.1272 ry=-2.0524 rz=-2.0554 rad; joints [-78.717, -44.993, 105.704, -61.467, 88.292, 5.922] deg; positionType=FIXED_POSITION; waypointPoseInFeatureCoordinates=(pos=(x=-0.22213279810283795, y=0.5429928607942448, z=-0.046020490685082405), rot=(x=0.12717824023039923, y=-2.0524184980685685, z=-2.0554068448244966)); name=Point_de_passag_54
      Waypoint blendRadius=0.05; cartesianAcceleration=1.2; cartesianSpeed=0.25; jointAcceleration=1.3962634015954636; jointSpeed=1.0471975511965976; nextMotionTime=2.0; stoppoint=true; useSharedBlendParameter=true; useSharedParameters=true; position=TCP in base x=-221.698 y=540.937 z=-54.117 mm, rx=0.1271 ry=-2.053 rz=-2.055 rad; joints [-78.719, -44.142, 105.934, -62.52, 88.294, 5.922] deg; positionType=FIXED_POSITION; waypointPoseInFeatureCoordinates=(pos=(x=-0.22169779398028377, y=0.540936684279263, z=-0.05411699580003387), rot=(x=0.12712563865135826, y=-2.0529878996076363, z=-2.0549769259995205)); name=Point_de_passag_55
      Waypoint blendRadius=0.05; cartesianAcceleration=1.2; cartesianSpeed=0.25; jointAcceleration=1.3962634015954636; jointSpeed=1.0471975511965976; nextMotionTime=2.0; stoppoint=true; useSharedBlendParameter=true; useSharedParameters=true; position=TCP in base x=-220.158 y=528.804 z=-53.42 mm, rx=0.1296 ry=-2.078 rz=-2.0313 rad; joints [-78.632, -45.114, 107.688, -61.952, 88.293, 5.922] deg; positionType=FIXED_POSITION; waypointPoseInFeatureCoordinates=(pos=(x=-0.22015789553627102, y=0.5288043377435323, z=-0.053420078544446456), rot=(x=0.12955647755320765, y=-2.0779553816467278, z=-2.031257330131183)); name=Point_de_passag_56
      Waypoint blendRadius=0.05; cartesianAcceleration=1.2; cartesianSpeed=0.25; jointAcceleration=1.3962634015954636; jointSpeed=1.0471975511965976; nextMotionTime=2.0; stoppoint=true; useSharedBlendParameter=true; useSharedParameters=true; position=TCP in base x=-206.325 y=530.415 z=-53.222 mm, rx=0.1042 ry=-2.0848 rz=-2.05 rad; joints [-80.053, -45.363, 108.408, -62.685, 88.294, 5.922] deg; positionType=FIXED_POSITION; waypointPoseInFeatureCoordinates=(pos=(x=-0.20632468785788477, y=0.5304146217066494, z=-0.05322241821281719), rot=(x=0.10416517014565908, y=-2.0847948523248463, z=-2.0499560696448382)); name=Point_de_passag_57
      Waypoint blendRadius=0.05; cartesianAcceleration=1.2; cartesianSpeed=0.25; jointAcceleration=1.3962634015954636; jointSpeed=1.0471975511965976; nextMotionTime=2.0; stoppoint=true; useSharedBlendParameter=true; useSharedParameters=true; position=TCP in base x=-207.531 y=539.592 z=-55.22 mm, rx=0.1025 ry=-2.039 rz=-2.0912 rad; joints [-80.093, -44.331, 107.401, -65.115, 88.294, 5.922] deg; positionType=FIXED_POSITION; waypointPoseInFeatureCoordinates=(pos=(x=-0.20753071492850722, y=0.5395917087675636, z=-0.055219628164308816), rot=(x=0.10245812906136402, y=-2.0390057032587956, z=-2.091195979959705)); name=Point_de_passag_58
      Waypoint blendRadius=0.05; cartesianAcceleration=1.2; cartesianSpeed=0.25; jointAcceleration=1.3962634015954636; jointSpeed=1.0471975511965976; nextMotionTime=2.0; stoppoint=true; useSharedBlendParameter=true; useSharedParameters=true; position=TCP in base x=-221.401 y=537.538 z=-55.153 mm, rx=0.1269 ry=-2.0253 rz=-2.0786 rad; joints [-78.681, -44.118, 106.858, -64.896, 88.303, 5.914] deg; positionType=FIXED_POSITION; waypointPoseInFeatureCoordinates=(pos=(x=-0.22140101643261081, y=0.5375375158389529, z=-0.055153071408574623), rot=(x=0.12686146374247875, y=-2.0253246214814355, z=-2.0785884529799357)); name=Point_de_passag_59
      Waypoint blendRadius=0.05; cartesianAcceleration=1.2; cartesianSpeed=0.25; jointAcceleration=1.3962634015954636; jointSpeed=1.0471975511965976; nextMotionTime=2.0; stoppoint=true; useSharedBlendParameter=true; useSharedParameters=true; position=TCP in base x=-220.246 y=529.965 z=-54.355 mm, rx=0.1284 ry=-2.0525 rz=-2.0544 rad; joints [-78.645, -44.824, 107.828, -63.733, 88.302, 5.914] deg; positionType=FIXED_POSITION; waypointPoseInFeatureCoordinates=(pos=(x=-0.22024606154509482, y=0.5299646898006728, z=-0.05435453969439623), rot=(x=0.12844427970352718, y=-2.052476818486931, z=-2.0543825592386042)); name=Point_de_passag_61
      Waypoint blendRadius=0.05; cartesianAcceleration=1.2; cartesianSpeed=0.25; jointAcceleration=1.3962634015954636; jointSpeed=1.0471975511965976; nextMotionTime=2.0; stoppoint=true; useSharedBlendParameter=true; useSharedParameters=true; position=TCP in base x=-210.436 y=531.583 z=-54.567 mm, rx=0.1108 ry=-2.0658 rz=-2.0603 rad; joints [-79.658, -44.96, 108.144, -63.655, 88.302, 5.914] deg; positionType=FIXED_POSITION; waypointPoseInFeatureCoordinates=(pos=(x=-0.2104357909804574, y=0.5315829560497437, z=-0.054567337868033285), rot=(x=0.11080414880507461, y=-2.0658088781786756, z=-2.06034478116537)); name=Point_de_passag_62
      Waypoint blendRadius=0.05; cartesianAcceleration=1.2; cartesianSpeed=0.25; jointAcceleration=1.3962634015954636; jointSpeed=1.0471975511965976; nextMotionTime=2.0; stoppoint=true; useSharedBlendParameter=true; useSharedParameters=true; position=TCP in base x=-219.597 y=533.239 z=-53.618 mm, rx=0.1262 ry=-2.0487 rz=-2.0598 rad; joints [-78.776, -44.714, 107.415, -63.68, 88.29, 5.914] deg; positionType=FIXED_POSITION; waypointPoseInFeatureCoordinates=(pos=(x=-0.21959735146789783, y=0.5332388105290958, z=-0.053617840042057975), rot=(x=0.12619587040185928, y=-2.048676484009864, z=-2.0598154842757124)); name=Point_de_passag_63
      Waypoint blendRadius=0.05; cartesianAcceleration=1.2; cartesianSpeed=0.25; jointAcceleration=1.3962634015954636; jointSpeed=1.0471975511965976; nextMotionTime=2.0; stoppoint=true; useSharedBlendParameter=true; useSharedParameters=true; position=TCP in base x=-211.206 y=536.662 z=-53.604 mm, rx=0.1105 ry=-2.0558 rz=-2.0693 rad; joints [-79.676, -44.712, 107.412, -63.694, 88.29, 5.914] deg; positionType=FIXED_POSITION; waypointPoseInFeatureCoordinates=(pos=(x=-0.2112060042072216, y=0.5366620468962878, z=-0.05360358444799081), rot=(x=0.11045269497356373, y=-2.0558333930439154, z=-2.0692685520928458)); name=Point_de_passag_64
